// TwinCAT 3 PLC project DMX_Plc
// ProgramVersion: 3.1.4026.17
// libraries:
//   Tc2_DMX, * (Beckhoff Automation GmbH)
//   Tc2_Standard, * (Beckhoff Automation GmbH)
//   Tc2_System, * (Beckhoff Automation GmbH)
// project tree:
//   DUTs/ DMX_Control.TcDUT, DMX_Status.TcDUT, DMX_Mode.TcDUT, Mover_13Ch.TcDUT
//   / PlcTask.TcTTO
//   POUs/ MAIN.TcPOU, ModeSwitch.TcPOU
// real-time tasks:
//   TASK PlcTask: cycle T#10ms, priority 20, ADS port 350
// I/O:
//   DEVICE Device 1 (EtherCAT), AmsNetId 10.200.106.16.2.1
//     Term 1 (EK1200) [EK1200-5000 EtherCAT Power supply (2A E-Bus)]
//       Term 2 (EL6851) [EL6851 DMX Master]
//       Term 3 (EL9011) [EL9011 End Terminal]
// variable links:
//   DMX_Plc/DMX_Plc Instance <-> Device 1 (EtherCAT)/Term 1 (EK1200)/Term 2 (EL6851)
//     PlcTask Inputs/MAIN.ST_EL6851InData_01/bCyclicTxDDisabled <-> DMX Status/Cyclic TxD disabled
//     PlcTask Inputs/MAIN.ST_EL6851InData_01/bDefaultDataSent <-> DMX Status/Default data sent
//     PlcTask Inputs/MAIN.ST_EL6851InData_01/bFrameSentToggle <-> DMX Status/Frame sent toggle
//     PlcTask Inputs/MAIN.ST_EL6851InData_01/bInputToggle <-> WcState/InputToggle
//     PlcTask Inputs/MAIN.ST_EL6851InData_01/bReceiveToggle <-> DMX Status/Receive toggle
//     PlcTask Inputs/MAIN.ST_EL6851InData_01/bTransmitAccepted <-> DMX Status/Transmit accepted
//     PlcTask Inputs/MAIN.ST_EL6851InData_01/bTxPDOToggle <-> DMX Status/TxPDO Toggle
//     PlcTask Inputs/MAIN.ST_EL6851InData_01/bWcState <-> WcState/WcState
//     PlcTask Inputs/MAIN.ST_EL6851InData_01/byStartCode <-> DMX Status/Start code
//     PlcTask Inputs/MAIN.ST_EL6851InData_01/stAdsAddr <-> InfoData/AdsAddr
//     PlcTask Inputs/MAIN.ST_EL6851InData_01/uiState <-> InfoData/State
//     PlcTask Inputs/MAIN.ST_EL6851InData_01/wChannelLength <-> DMX Status/Channel length
//     PlcTask Outputs/MAIN.Mover1/Blue <-> DMX Channel 1-64/Channel 10
//     PlcTask Outputs/MAIN.Mover1/CH12 <-> DMX Channel 1-64/Channel 12
//     PlcTask Outputs/MAIN.Mover1/CH13 <-> DMX Channel 1-64/Channel 13
//     PlcTask Outputs/MAIN.Mover1/Dimming <-> DMX Channel 1-64/Channel 6
//     PlcTask Outputs/MAIN.Mover1/Green <-> DMX Channel 1-64/Channel 9
//     PlcTask Outputs/MAIN.Mover1/Pan <-> DMX Channel 1-64/Channel 1
//     PlcTask Outputs/MAIN.Mover1/PanFine <-> DMX Channel 1-64/Channel 2
//     PlcTask Outputs/MAIN.Mover1/PanTiltSpeed <-> DMX Channel 1-64/Channel 5
//     PlcTask Outputs/MAIN.Mover1/Red <-> DMX Channel 1-64/Channel 8
//     PlcTask Outputs/MAIN.Mover1/Strobe <-> DMX Channel 1-64/Channel 7
//     PlcTask Outputs/MAIN.Mover1/Tilt <-> DMX Channel 1-64/Channel 3
//     PlcTask Outputs/MAIN.Mover1/TiltFine <-> DMX Channel 1-64/Channel 4
//     PlcTask Outputs/MAIN.Mover1/White <-> DMX Channel 1-64/Channel 11
//     PlcTask Outputs/MAIN.ST_EL6851OutData_01/bDisableCyclicTxD <-> DMX Control/Disable cyclic TxD
//     PlcTask Outputs/MAIN.ST_EL6851OutData_01/bSendDefaultData <-> DMX Control/Send default data
//     PlcTask Outputs/MAIN.ST_EL6851OutData_01/bTransmitRequest <-> DMX Control/Transmit request
//     PlcTask Outputs/MAIN.ST_EL6851OutData_01/byStartCode <-> DMX Control/Start code
//     PlcTask Outputs/MAIN.ST_EL6851OutData_01/wChannelLength <-> DMX Control/Channel length

CONFIGURATION DMX_Plc
    RESOURCE PLC ON TwinCAT3
        TASK PlcTask(INTERVAL := T#10ms, PRIORITY := 20);
        PROGRAM MAIN WITH PlcTask : MAIN;
    END_RESOURCE
END_CONFIGURATION

// ---- DUTs/DMX_Control.TcDUT
TYPE DMX_Control :
STRUCT
	TransmitRequest : BIT;
	DisableCyclicTxD : BIT;
	SendDefaultData : BIT;
	ChannelLength : UINT;
	StartCode : USINT;
END_STRUCT
END_TYPE

// ---- DUTs/DMX_Status.TcDUT
TYPE DMX_Status :
STRUCT
	TransmitAccepted : BIT;
	RecieveToggle : BIT;
	CyclicTxD_Disabled : BIT;
	DefaultDataSent : BIT;
	FrameSentToggle : BIT;
	TxPdoToggle : BIT;
	ChannelLength : UINT;
	StartCode : USINT;
END_STRUCT
END_TYPE

// ---- DUTs/DMX_Mode.TcDUT
{attribute 'qualified_only'}
{attribute 'strict'}
{attribute 'to_string'}
TYPE DMX_Mode :
(
	INIT := 0,
	MODE_ADDRESS,
	MODE_DMX_DISCOVERY,
	MODE_SET_ADDRESS,
	MODE_OPTICAL_FEEDBACK,
	ERROR
);
END_TYPE

// ---- DUTs/Mover_13Ch.TcDUT
TYPE Mover_13Ch :
STRUCT
	Pan : BYTE;
	PanFine : BYTE;
	Tilt : BYTE;
	TiltFine : BYTE;
	PanTiltSpeed : BYTE;
	Dimming : BYTE;
	Strobe : BYTE;
	Red : BYTE;
	Green : BYTE;
	Blue : BYTE;
	White : BYTE;
	CH12 : BYTE; //0-30 = No Function, 31-127 = Auto 1, 127-249 = Auto 2, 250-255 = Sound Mode
	CH13 : BYTE; //0-149 = No Function, 150-200 = Reset, 201-255 = No Function
END_STRUCT
END_TYPE

// ---- POUs/MAIN.TcPOU
PROGRAM MAIN

VAR
	
	eDMX_Mode : DMX_Mode;
	
	//Var to select the Mode the DMX should operate in
	// 0 = ADDRESS Mode, 1 = RDM Mode, 2 = DMX Address Set, 3 = Optical Feedback
	iModeSelect : INT := 1; 


	//DMX Fuction Blocks
	FB_DMXDiscovery512_01: FB_DMXDiscovery512;
	DMX_CommandBuffer:ST_DMXCommandBuffer;
	FB_EL6851CommunicationEx_01: FB_EL6851CommunicationEx;
	ST_EL6851InData_01 AT %I* : ST_EL6851InDataEx;
	ST_EL6851OutData_01 AT %Q*: ST_EL6851OutData;
	ProcessData : ARRAY [1..512] OF BYTE; 
	
	//Mover Control Structure
	Mover1 AT %Q* : Mover_13Ch;
	
	FixtureChLength : UINT := 13;
	
	
END_VAR

CASE eDMX_Mode OF
	//Initialize state
	DMX_Mode.INIT:
		//Checks for errors then moves to the mode selected with iModeSelect
		IF NOT FB_EL6851CommunicationEx_01.bError AND NOT FB_DMXDiscovery512_01.bError THEN
			eDMX_Mode := ModeSwitch(iModeSelect);
		END_IF
		
	//Cyclic Writing to DMX Addresses
	DMX_Mode.MODE_ADDRESS:
		FB_EL6851CommunicationEx_01.bSetCycleMode := TRUE;
		FB_EL6851CommunicationEx_01.bEnableSendingData := TRUE;
		FB_EL6851CommunicationEx_01.uiDataLength := FixtureChLength;
		
		//Exit the MODE_ADDRESS state to change to a different mode
		IF NOT FB_DMXDiscovery512_01.bBusy THEN
			FB_DMXDiscovery512_01.bStart := FALSE;
			eDMX_Mode := ModeSwitch(iModeSelect);
		END_IF
		
	//DMX Discovery - Non cyclic 	
	DMX_Mode.MODE_DMX_DISCOVERY:
		FB_EL6851CommunicationEx_01.bSetCycleMode := FALSE;
		FB_EL6851CommunicationEx_01.bSetCycleMode := FALSE;
		FB_DMXDiscovery512_01.bStart := TRUE;
		FB_DMXDiscovery512_01.dwOptions := DMX_OPTION_COMPLETE_NEW_DISCOVERY;
		
		//Exit the MODE_DMX_Discovery State to change to a different mode
		IF NOT FB_DMXDiscovery512_01.bBusy THEN
			eDMX_Mode := ModeSwitch(iModeSelect);
		END_IF
	
	//DMX Set Addresses - Non cyclic 	
	DMX_Mode.MODE_SET_ADDRESS:
		FB_EL6851CommunicationEx_01.bSetCycleMode := FALSE;
		FB_EL6851CommunicationEx_01.bSetCycleMode := FALSE;
		FB_DMXDiscovery512_01.bStart := TRUE;
		FB_DMXDiscovery512_01.dwOptions := DMX_OPTION_SET_START_ADDRESS;
		
		//Exit the MODE_DMX_Discovery State to change to a different mode
		IF NOT FB_DMXDiscovery512_01.bBusy THEN
			FB_DMXDiscovery512_01.bStart := FALSE;
			eDMX_Mode := ModeSwitch(iModeSelect);
		END_IF
		
	//DMX Optical Feedback - Non cyclic 	
	DMX_Mode.MODE_OPTICAL_FEEDBACK:
		FB_EL6851CommunicationEx_01.bSetCycleMode := FALSE;
		FB_EL6851CommunicationEx_01.bSetCycleMode := FALSE;
		FB_DMXDiscovery512_01.bStart := TRUE;
		FB_DMXDiscovery512_01.dwOptions := DMX_OPTION_OPTICAL_FEEDBACK;
		
		//Exit the MODE_DMX_Discovery State to change to a different mode
		IF NOT FB_DMXDiscovery512_01.bBusy THEN
			FB_DMXDiscovery512_01.bStart := FALSE;
			eDMX_Mode := ModeSwitch(iModeSelect);
		END_IF
	
	DMX_Mode.ERROR:


END_CASE;

//Call FB's
FB_EL6851CommunicationEx_01(
	stEL6851InData:= ST_EL6851InData_01, 
	stEL6851OutData:= ST_EL6851OutData_01, 
	stCommandBuffer:= DMX_CommandBuffer, 
	arrProcessData:= ProcessData);
	
FB_DMXDiscovery512_01(
	stCommandBuffer:= DMX_CommandBuffer);

END_PROGRAM

// ---- POUs/ModeSwitch.TcPOU
FUNCTION ModeSwitch : DMX_Mode
VAR_INPUT
	Target	: INT;
END_VAR
VAR
	eMode : DMX_Mode;
END_VAR


IF Target = 0 THEN
	eMode := DMX_Mode.INIT;
ELSIF Target = 1 THEN
	eMode := DMX_Mode.MODE_ADDRESS;
ELSIF Target = 2 THEN
	eMode := DMX_Mode.MODE_DMX_DISCOVERY;
ELSIF Target = 3 THEN
	eMode := DMX_Mode.MODE_SET_ADDRESS;
ELSIF Target = 4 THEN
	eMode := DMX_Mode.MODE_OPTICAL_FEEDBACK;
END_IF

ModeSwitch := eMode;

END_FUNCTION
